INTERFACE I_McAxis

PROPERTY AxisRef : reference to AXIS_REF
GET
END_GET
END_PROPERTY

END_INTERFACE

(* stored: Version 1.1.0.1, ProductVersion 3.1.4024.12
   Itf I_McAxis: Id {df9f672e-6c08-07db-39bc-3fcca419c0c5}
   Folder properties: Id {c3aa66e4-adb2-0576-2fa7-bb2e1744bc40}
   Property AxisRef: Id {5b5f341e-5598-0c1b-0e07-a2e86f8ec7a8}
   Get Get: Id {e308e6f3-b4af-0894-0c9f-f1d325a62694} *)
